// TwinCAT 3 PLC project LightFunctions
// ProgramVersion: 3.1.4023.0
// libraries:
//   CmpBitmapPool, * (System)
//   Tc2_BABasic, * (Beckhoff Automation GmbH)
//   Tc2_Standard, * (Beckhoff Automation GmbH)
//   Tc2_System, * (Beckhoff Automation GmbH)
//   Tc2_TcpIp, * (Beckhoff Automation GmbH)
//   Tc2_Utilities, * (Beckhoff Automation GmbH)
//   Tc3_Module, * (Beckhoff Automation GmbH)
//   VisuSymbols,3.5.10.0,System
// project tree:
//   DUTs/ E_State.TcDUT (not stored)
//   / GlobalTextList.TcGTLO, PlcTask.TcTTO, Visualization Manager.TcVMO (not stored)
//   POUs/ FB_TcpServer.TcPOU, FnR_Switch.TcPOU, MAIN.TcPOU, Pedal.TcPOU (not stored)
//   VISUs/ ImagePool.TcIPO (not stored), Visualization.TcVIS
// real-time tasks:
//   TASK PlcTask: cycle T#10ms, priority 20, ADS port 350

CONFIGURATION LightFunctions
    RESOURCE PLC ON TwinCAT3
        TASK PlcTask(INTERVAL := T#10ms, PRIORITY := 20);
        PROGRAM MAIN WITH PlcTask : MAIN;
    END_RESOURCE
END_CONFIGURATION

// ---- POUs/MAIN.TcPOU
PROGRAM MAIN
VAR
	fbTcpServer 	: FB_TcpServer;
	SrvNetId		: STRING := '';
	ServerAddress 	: STRING := '';
	ServerPort 		: UDINT := 24100;
	
	sResponse		: STRING;
	sCommand		: STRING;
	bBusy			: BOOL;
	err				: BOOL;
	errid			: UDINT;
	
//	blinkLeft : BOOL;
//	blinkRight : BOOL;
//	lightFront : BOOL;
//	lightRear : BOOL;
//	lightBrake : BOOL;

	LightsFront   : BOOL;
	LightsRear 	: BOOL;
	LightsBrake	: BOOL;
	LightsReverse : BOOL;
    BlinkerLeft     : BOOL;
    BlinkerRight    : BOOL;
	
	test: STRING;
END_VAR

fbTcpServer(
	NetId:= SrvNetId, 
	ServerAdr:= ServerAddress, 
	ServerPort:= ServerPort, 
	sSend := sResponse,
	sReceive=> sCommand, 
	bBusy=> bBusy, 
	err=> err, 
	errid=> errid);
	
	sResponse := sCommand;
	
	Ping();
	Pedal();

//IF sCommand = 'blinker:left' THEN
//	blinkLeft := TRUE;
//ELSIF sCommand = 'blinker:right' THEN
//	blinkRight := TRUE;
//ELSE
//	blinkLeft := FALSE;
//	blinkRight := FALSE;
//END_IF

IF sCommand = 'blon' THEN	//blinker left on
    BlinkerLeft    := TRUE;
    BlinkerRight   := FALSE;
ELSIF sCommand = 'bloff' THEN	//blinker left off
    BlinkerLeft    := FALSE;
    BlinkerRight := FALSE;
ELSIF sCommand = 'bron' THEN	//blinker right on
    BlinkerRight   := TRUE;
    BlinkerLeft    := FALSE;
ELSIF sCommand = 'broff' THEN	//blinker right off
    BlinkerRight  := FALSE;
    BlinkerLeft   := FALSE;
ELSIF sCommand = 'lon' THEN //lights on
	LightsFront := TRUE;
	LightsRear := TRUE;
ELSIF sCommand = 'loff' THEN	//lights off
	LightsFront := FALSE;
	LightsRear := FALSE;
ELSIF sCommand = 'ron' THEN	//reverse light on
	LightsReverse := TRUE;
ELSIF sCommand = 'roff' THEN	//reverse light off
	LightsReverse := FALSE;
ELSIF sCommand = 'bon' THEN	//reverse light on
	LightsBrake := TRUE;
ELSIF sCommand = 'boff' THEN	//reverse light off
	LightsBrake := FALSE;
ELSE
    BlinkerRight := FALSE;
    BlinkerLeft  := FALSE;

END_IF

END_PROGRAM

// ---- POUs/FB_TcpServer.TcPOU
FUNCTION_BLOCK FB_TcpServer
VAR_INPUT
	NetId				: STRING; 	(* Server AmsNetId *)
	ServerAdr 			: STRING;	(* Server IP address *)
	ServerPort 			: UDINT;	(* Server port number *)
	sSend 				: STRING;	(* String to be sent *)
END_VAR
VAR_OUTPUT
	sReceive			: STRING;	(* String received *)
	bBusy				: BOOL;
	err					: BOOL;
	errid				: UDINT;
END_VAR
VAR
	fbSocketCloseAll	: FB_SocketCloseAll :=  ( sSrvNetID := '', tTimeout := DEFAULT_ADS_TIMEOUT );
	bCloseAll			: BOOL := TRUE;
		
	Timeout 			: TIME := T#10S;
	fbSocketListen		: FB_SocketListen := (bExecute := TRUE);
	fbSocketReceive		: FB_SocketReceive;
	fbSocketAccept		: FB_SocketAccept;
	fbSocketSend 		: FB_SocketSend;
	hListen				: T_HSOCKET;
	hSocket				: T_HSOCKET;
    
	bConnAccepted		: BOOL;            	
	RxBuffer			: STRING;
	state				: E_State;
           	
	timer				: TON;
	
	fbLocalTime : FB_LocalSystemTime;
	iPreviousTime : WORD := 0;
	SafetyTriggerd : BOOL;
	
END_VAR

//https://github.com/vancassa/TwinCAT_TCP_IP_Server/tree/master/Examples/TwinCAT_Program

IF bCloseAll THEN (*On PLC reset or program download close all old connections *)
	bCloseAll := FALSE;
	fbSocketCloseAll( bExecute:= TRUE );
ELSE
	fbSocketCloseAll( bExecute:= FALSE );
END_IF

IF sSend = '' THEN
	sSend := 'Default response';
END_IF
				
timer(IN:= , PT:= T#500MS, Q=> , ET=> );

fbLocalTime(
	sNetId := ,
	bEnable := TRUE,
	dwCycle := 10,
	dwOpt := ,
	tTimeout := DEFAULT_ADS_TIMEOUT,
);

	IF fbLocalTime.systemTime.wMilliseconds - iPreviousTime >= 200 THEN	
		SafetyTriggerd := TRUE;	
	END_IF
	
	IF MAIN.sCommand > '' THEN
		iPreviousTime := fbLocalTime.systemTime.wMilliseconds;
		
	END_IF
 
fbSocketListen(
		sSrvNetId:= NetId, 
		sLocalHost:= ServerAdr, 
		nLocalPort:= ServerPort, 
		bExecute:= , 
		tTimeout:= Timeout, 
		bBusy=> bBusy, 
		bError=> err, 
		nErrId=> errid, 
		hListener=> hListen);

fbSocketAccept(
		sSrvNetId:= NetId, 
		hListener:= hListen, 
		bExecute:= , 
		tTimeout:= Timeout, 
		bAccepted=> bConnAccepted, 
		bBusy=> bBusy, 
		bError=> err, 
		nErrId=> errid, 
		hSocket=> hSocket);
	
fbSocketSend(
		sSrvNetId:= NetId, 
		hSocket:= hSocket, 
		cbLen:= LEN(sSend), 
		pSrc:= ADR(sSend), 
		bExecute:= , 
		tTimeout:= Timeout, 
		bBusy=> bBusy, 
		bError=> err, 
		nErrId=> errid);

fbSocketReceive(
		sSrvNetId:= NetId, 
		hSocket:= hSocket, 
		cbLen:= SIZEOF(RxBuffer), 
		pDest:= ADR(RxBuffer), 
		bExecute:= , 
		tTimeout:= Timeout, 
		bBusy=> bBusy, 
		bError=> err, 
		nErrId=> errid, 
		nRecBytes=> );
		
CASE state OF
	E_State.STATE_INIT:
		//Open the port
		fbSocketListen.bExecute := TRUE;
		state := E_State.STATE_CONNECTING;
		
		
	E_State.STATE_CONNECTING:
		fbSocketListen.bExecute := FALSE;
		//Accept incoming connection every half a second
		IF NOT fbSocketListen.bBusy AND NOT fbSocketListen.bError THEN
			fbSocketAccept.bExecute := FALSE;
			timer.IN := TRUE;
	
			IF bConnAccepted THEN
				fbSocketReceive.bExecute := TRUE;
				state := E_State.STATE_RECEIVING_DATA;
			ELSIF timer.Q THEN
				fbSocketAccept.bExecute := TRUE;
				timer.IN := FALSE;
			END_IF
		END_IF
	
		
	E_State.STATE_RECEIVING_DATA:
		fbSocketReceive.bExecute := FALSE;
		
		IF NOT fbSocketReceive.bBusy AND NOT fbSocketReceive.bError THEN
			IF fbSocketReceive.nRecBytes = 0 THEN
				//if there's no data received, reset the fbSocketReceive
				fbSocketReceive.bExecute := TRUE;
			ELSE
				MEMSET(ADR(sReceive),0,SIZEOF(sReceive));
				MEMCPY(ADR(sReceive), fbSocketReceive.pDest, fbSocketReceive.nRecBytes);
				

				fbSocketSend.bExecute := TRUE;
				state := E_State.STATE_SENDING_DATA;
			END_IF
		END_IF
	
		
	E_State.STATE_SENDING_DATA:
		fbSocketSend.bExecute := FALSE;
		
		IF NOT fbSocketSend.bBusy AND NOT fbSocketSend.bError THEN 
				fbSocketReceive.bExecute := TRUE;
				state := E_State.STATE_RECEIVING_DATA;
		END_IF
END_CASE

END_FUNCTION_BLOCK

// ---- POUs/FnR_Switch.TcPOU
PROGRAM FnR_Switch
VAR
	qFNR : BOOL; //0 = user control, 1 = PLC controlled FNR
	qFNRDir : BOOL; //Sets direction 0 = reverse, 1 = forward
END_VAR

//Program to select what direction the car should go
IF MAIN.sCommand = 'Forward' THEN
	qFNR := TRUE;
	qFNRDir := TRUE;
ELSIF MAIN.sCommand = 'Reverse' THEN
	qFNR := TRUE;
	qFNRDir := FALSE;
ELSIF Main.sCommand = 'Manual' THEN //supposed to be manual mode
	qFNR := FALSE;
	qFNRDir := FALSE; //This one doesn't really matter
END_IF

END_PROGRAM

// ---- VISUs/Visualization.TcVIS
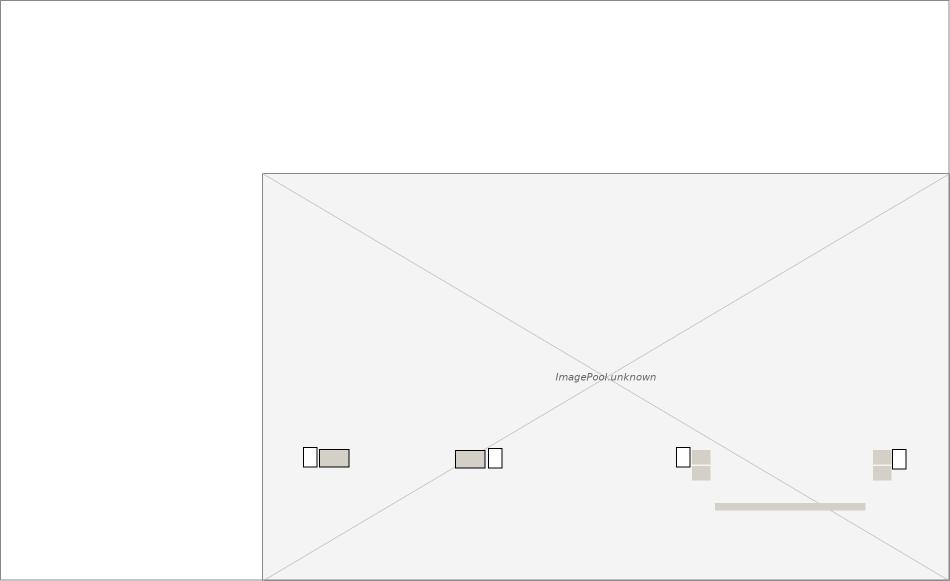
VISUALIZATION Visualization  // 950x581
    Image (262,173 688x408), image: ImagePool.unknown
    RoundedRectangle (488,448 14x20), colour toggle: MAIN.BlinkerLeft
    RoundedRectangle (303,447 14x20), colour toggle: MAIN.BlinkerRight
    RoundedRectangle (455,450 30x18), colour toggle: MAIN.LightsFront
    RoundedRectangle (676,447 14x20), colour toggle: MAIN.BlinkerLeft
    RoundedRectangle (892,449 14x20), colour toggle: MAIN.BlinkerRight
    RoundedRectangle (319,449 30x18), colour toggle: MAIN.LightsFront
    RoundedRectangle (692,450 18x14), colour toggle: MAIN.LightsRear
    RoundedRectangle (692,466 18x14), colour toggle: MAIN.LightsBrake
    RoundedRectangle (873,450 18x14), colour toggle: MAIN.LightsRear
    RoundedRectangle (873,466 18x14), colour toggle: MAIN.LightsBrake
    RoundedRectangle (715,503 150x7), colour toggle: MAIN.LightsReverse
END_VISUALIZATION
